PROGRAM AutomaticLogic_1
VAR
	Compressor1: Compressor;
	Tracking1: TrackingLogic;
	AutoCtrl: AutomationControl_1;
	Id_counter: CTU;
	Sensor1_FTrig: F_TRIG;
	lastP_trig: R_TRIG;
	limit1_trig: R_TRIG;
	
	activate: BOOL;
	vert_p: Vertical_process;
END_VAR

//AutoCtrl(piston1for := FALSE, piston1back := FALSE, piston2for := FALSE, piston2back := FALSE, pistonVert := FALSE, motorCon := FALSE, motorRotate := FALSE);
AutoCtrl();
Compressor1(switch:= GVL.Switch);
Tracking1();
Sensor1_FTrig(CLK:= GVL.Sensor1);
Id_counter();
lastP_trig(CLK := GVL.Sensor2);
Id_counter.CU := Sensor1_FTrig.Q;
limit1_trig(CLK:= GVL.Limit1);

vert_p(activate:= activate);


IF GVL.Switch = FALSE THEN
	
	//Init of Pieces
	IF Sensor1_FTrig.Q = TRUE THEN
		GVL.Position[0].Piece.Id := TO_INT(Id_counter.CV);
		GVL.Position[0].Piece.Recipe := 1;
		GVL.Position[0].Occupied := TRUE;
	END_IF
	
	// pushing from position 0
	IF (NOT GVL.Position[1].Occupied AND NOT AutoCtrl.motorRotate AND GVL.Position[0].Occupied) THEN
	AutoCtrl.piston1back := FALSE;	
	AutoCtrl.piston1for := TRUE;
		IF (GVL.Sensor1) THEN
			AutoCtrl.piston1for := FALSE;
			AutoCtrl.piston1back := TRUE;
			GVL.Position[0].Done := TRUE;
		END_IF
	END_IF

	// rotating table
	IF ((GVL.Position[1].Occupied AND NOT GVL.Position[2].Occupied AND NOT GVL.Position[3].Occupied) OR (NOT GVL.Position[1].Occupied AND (GVL.Position[2].Occupied AND GVL.Position[2].Processed) AND NOT GVL.Position[3].Occupied) OR (GVL.Position[1].Occupied AND (GVL.Position[2].Occupied AND GVL.Position[2].Processed) AND NOT GVL.Position[3].Occupied)) THEN
		AutoCtrl.motorRotate := TRUE;
		IF (GVL.Position[1].Occupied AND NOT GVL.Position[2].Occupied AND NOT GVL.Position[3].Occupied) THEN
			IF (GVL.Limit1) THEN
				AutoCtrl.motorRotate := FALSE;
				GVL.Position[1].Done := TRUE;
			END_IF	
		END_IF
		IF (NOT GVL.Position[1].Occupied AND (GVL.Position[2].Occupied AND GVL.Position[2].Processed)) THEN
			IF (GVL.Limit2) THEN
				AutoCtrl.motorRotate := FALSE;
				GVL.Position[2].Done := TRUE;
			END_IF
		END_IF
		IF (GVL.Position[1].Occupied AND (GVL.Position[2].Occupied AND GVL.Position[2].Processed) AND NOT GVL.Position[3].Occupied) THEN
			IF (GVL.Limit2) THEN
				AutoCtrl.motorRotate := FALSE;
				GVL.Position[2].Done := TRUE;
				IF (NOT GVL.Position[2].Done) THEN
					GVL.Position[1].Done := TRUE;
				END_IF
			END_IF
		END_IF
		
	END_IF
	
	// processing
	IF (GVL.Position[2].Occupied AND NOT GVL.Position[2].Processed) THEN
		IF (GVL.Position[2].Piece.Processed <= GVL.Position[2].Piece.Id + 1) THEN
			activate := TRUE;
			IF (vert_p.done) THEN
				//GVL.Position[2].Piece.Processed := GVL.Position[2].Piece.Processed + 1;
				activate := FALSE;
				IF (GVL.Position[2].Piece.Processed >= GVL.Position[2].Piece.Id +1) THEN
					GVL.Position[2].Processed := TRUE;
					//GVL.Position[2].Done := TRUE;
				END_IF
			END_IF
		END_IF
	END_IF
	
	// Piston 2
	IF (GVL.Position[3].Occupied AND NOT GVL.Position[4].Occupied) THEN
		
		AutoCtrl.piston2for := FALSE;
		AutoCtrl.piston2back := TRUE;	
		IF (NOT GVL.Limit2) THEN
			AutoCtrl.piston2back := FALSE;
			AutoCtrl.piston2for := TRUE;
			GVL.Position[3].Done := TRUE;
		END_IF
	END_IF
	
	// motorCon
	IF (GVL.Position[4].Occupied AND NOT GVL.Position[5].Occupied) THEN
		AutoCtrl.motorCon := TRUE;
		IF (NOT GVL.Sensor2) THEN
			AutoCtrl.motorCon := FALSE;
			GVL.Position[4].Done := TRUE;
		END_IF
	END_IF
	
	// LaSt position
	IF (lastP_trig.Q) THEN
		GVL.Position[5].Done := TRUE;
	END_IF

	
END_IF

END_PROGRAM

(* stored: Version 1.1.0.1, ProductVersion 3.1.4024.12
   POU AutomaticLogic_1: Id {4cb8fbca-d5f6-4ba6-89b1-66d5dda03017}, SpecialFunc None *)
